FUNCTION_BLOCK EnhancedAdapter2 (* Basic FB with empty ECC *)
  (* Standard: 61499-2 *)
  (* Version 1.0, 2023-03-07, AK115394 *)
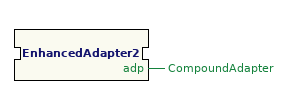
  PLUGS
    adp : CompoundAdapter;
  END_PLUGS
  EC_STATES
    START; (* Initial State *)
  END_STATES
END_FUNCTION_BLOCK
